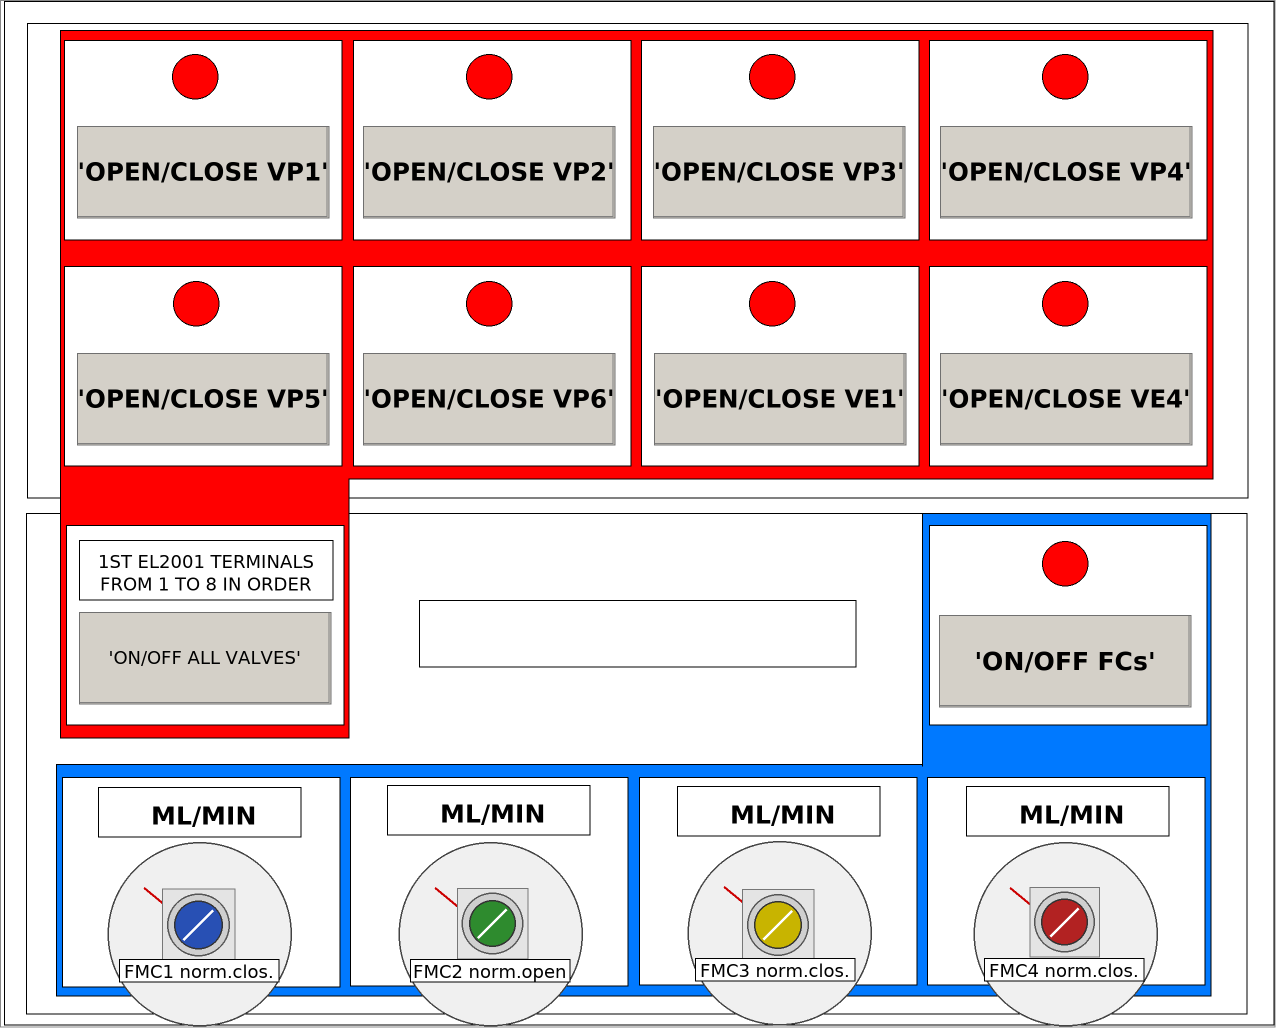
VISUALIZATION Visualization_1  // 1276x1028
    Rectangle (4,1 1270x1024)
    Rectangle (26,513 1221x501)
    Rectangle (56,764 1155x232)
    Rectangle (27,23 1221x475)
    RoundedRectangle (350,777 278x209)
    RoundedRectangle (62,777 278x210)
    RoundedRectangle (927,777 278x208)
    RoundedRectangle (639,777 278x208)
    Meter180 (104,842 191x184), value: MAIN.meter1, style: Meter-Meter180-Blue, scale format: %.1f, scale 0..500
    Potentiometer360 (162,886 73x78), variable: io.UI1_REF, style: Potentiometer-Potentiometer360-Blue, scale 0..500
        p2431819421: Outside
    Meter180 (395,842 191x184), value: MAIN.meter2, style: Meter-Meter180-Green, scale format: %.1f, scale 0..500
    Potentiometer360 (454,888 77x71), variable: io.UI2_REF, style: Potentiometer-Potentiometer360-Green, scale 0..500
        p2431819421: Outside
    Meter180 (684,841 191x184), value: MAIN.meter3, style: Meter-Meter180-Yellow, scale format: %.1f, scale 0..500
    Potentiometer360 (742,885 72x80), variable: io.UI3_REF, style: Potentiometer-Potentiometer360-Yellow, scale 0..500
        p2431819421: Outside
    Meter180 (970,842 191x184), value: MAIN.meter4, style: Meter-Meter180-Red, scale format: %.1f, scale 0..500
    Potentiometer360 (1029,887 71x70), variable: io.UI4_REF, style: Potentiometer-Potentiometer360-Red, scale 0..500
        p2431819421: Outside
    RoundedRectangle (98,787 203x50), text variable: meter1
    Textfield (123,795 162x41), "ML/MIN", text variable: MAIN.meter1
    RoundedRectangle (387,785 203x50)
    Textfield (412,793 162x41), "ML/MIN", text variable: MAIN.meter2
    RoundedRectangle (677,786 203x50)
    Textfield (702,794 162x41), "ML/MIN", text variable: MAIN.meter3
    RoundedRectangle (966,786 203x50)
    Textfield (991,794 162x41), "ML/MIN", text variable: MAIN.meter4
    RoundedRectangle (419,600 437x67)
    Label (392,588 495x92), "FLOW-COMMAND TOOL 2020"
    Rectangle (922,513 289x253)
    RoundedRectangle (929,525 278x200)
    Ellipse (1042,541 46x45), colour toggle: IO.fx1_REF
    Button (939,615 252x92), "'ON/OFF FCs'"
        OnMouseClick: toggle IO.fx1_REF
        OnMouseClick: toggle IO.fx2_REF
        OnMouseClick: toggle IO.fx3_REF
        OnMouseClick: toggle IO.fx4_REF
        OnMouseClick: toggle IO.fx5_REF
        OnMouseClick: toggle IO.fx6_REF
        OnMouseClick: toggle IO.fx7_REF
        OnMouseClick: toggle IO.fx8_REF
    Rectangle (60,477 289x261)
    Ellipse (181,536 46x45), colour toggle: IO.erikoismuuttujaSum
    RoundedRectangle (66,525 278x200)
    Button (79,612 252x92), "'ON/OFF ALL VALVES'"
        OnMouseClick: toggle IO.erikoismuuttujaSum
    Rectangle (60,30 1153x449)
    RoundedRectangle (353,266 278x200)
    RoundedRectangle (64,266 278x200)
    RoundedRectangle (353,40 278x200)
    RoundedRectangle (64,40 278x200)
    Ellipse (172,54 46x45), colour toggle: IO.r1_REF
    Button (77,126 252x92), "'OPEN/CLOSE VP1'"
        OnMouseClick: toggle IO.r1_REF
    Ellipse (466,54 46x45), colour toggle: IO.r2_REF
    Button (363,126 252x92), "'OPEN/CLOSE VP2'"
        OnMouseClick: toggle IO.r2_REF
    Ellipse (173,281 46x45), colour toggle: IO.r5_REF
    Button (77,353 252x92), "'OPEN/CLOSE VP5'"
        OnMouseClick: toggle IO.r5_REF
    Ellipse (466,281 46x45), colour toggle: IO.r6_REF
    Button (363,353 252x92), "'OPEN/CLOSE VP6'"
        OnMouseClick: toggle IO.r6_REF
    RoundedRectangle (929,266 278x200)
    RoundedRectangle (641,266 278x200)
    RoundedRectangle (929,40 278x200)
    RoundedRectangle (641,40 278x200)
    Ellipse (749,54 46x45), colour toggle: IO.r3_REF
    Button (653,126 252x92), "'OPEN/CLOSE VP3'"
        OnMouseClick: toggle IO.r3_REF
    Ellipse (1042,54 46x45), colour toggle: IO.r4_REF
    Button (940,126 252x92), "'OPEN/CLOSE VP4'"
        OnMouseClick: toggle IO.r4_REF
    Ellipse (749,281 46x45), colour toggle: IO.v1_REF
    Button (654,353 252x92), "'OPEN/CLOSE VE1'"
        OnMouseClick: toggle IO.v1_REF
    Ellipse (1042,281 46x45), colour toggle: IO.v2_REF
    Button (940,353 252x92), "'OPEN/CLOSE VE4'"
        OnMouseClick: toggle IO.v2_REF
    Rectangle (61,468 287x41)
    Rectangle (923,735 287x41)
    RoundedRectangle (119,959 160x23), text variable: meter1
    Textfield (120,963 158x18), "FMC1 norm.clos.", text variable: MAIN.meter3
    RoundedRectangle (410,959 160x23), text variable: meter1
    Textfield (411,963 158x18), "FMC2 norm.open", text variable: MAIN.meter3
    RoundedRectangle (695,958 160x23), text variable: meter1
    Textfield (696,962 158x18), "FMC3 norm.clos.", text variable: MAIN.meter3
    RoundedRectangle (984,958 160x23), text variable: meter1
    Textfield (985,962 158x18), "FMC4 norm.clos.", text variable: MAIN.meter3
    RoundedRectangle (79,540 254x60), text variable: meter1
    Textfield (80,549 252x48), "1ST EL2001 TERMINALS FROM 1 TO 8 IN ORDER", text variable: MAIN.meter3
END_VISUALIZATION

(* stored: Version 1.1.0.1, ProductVersion 3.1.4024.0
   Visu Visualization_1: Id {92402780-3208-4360-9dcb-7b60ec972095} *)
